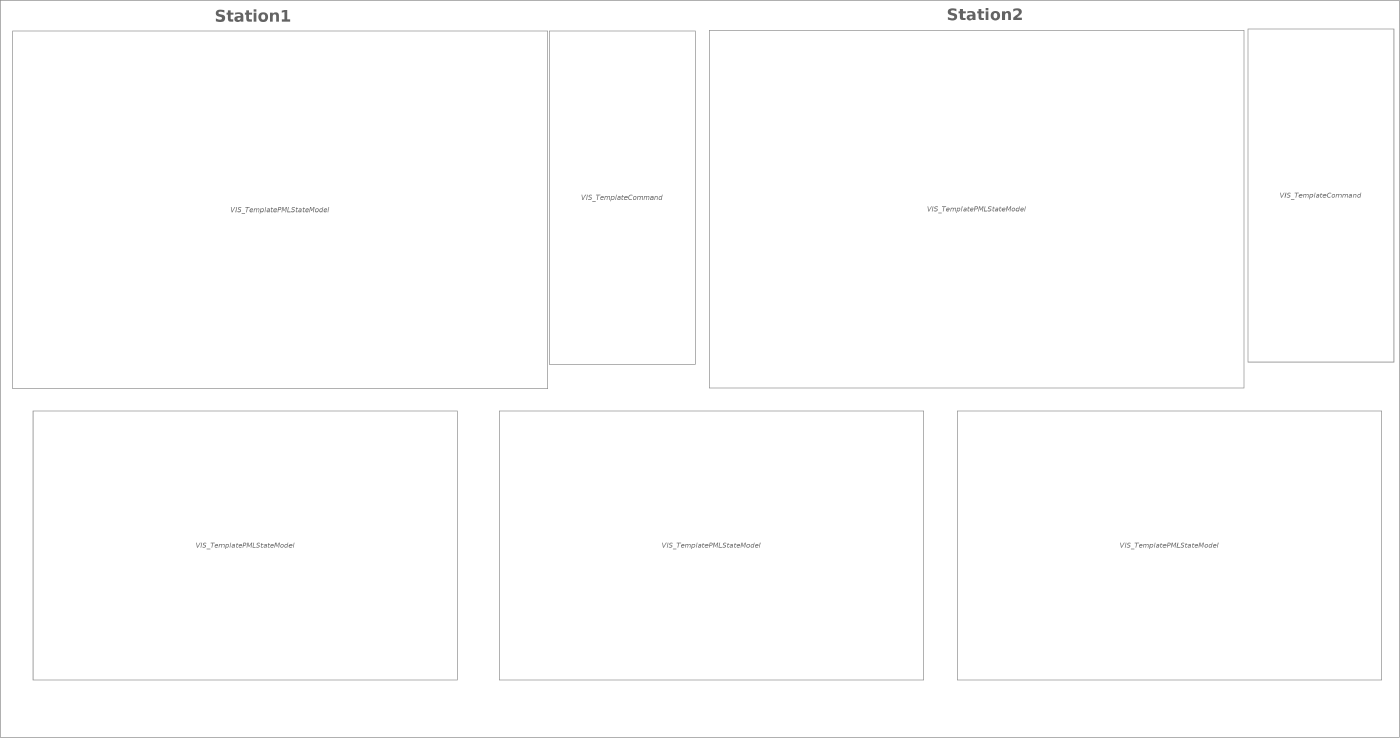
VISUALIZATION visu_2sys  // 2048x1080
    Frame (803,45 214x488)
        shows VIS_TemplateCommand(eModeCommand := GVL.PackTags.Command.UnitMode, eStateCommand := GVL.PackTags1.Command.CntrlCmd, eModeStatus := GVL.PackTags.Status.UnitModeCurrent, eStateStatus := GVL.PackTags1.Status.StateCurrent, bModeChangeReq := GVL.PackTags.Command.UnitModeChangeRequest)
    Frame (1825,42 214x488)
        shows VIS_TemplateCommand(eModeCommand := GVL.PackTags.Command.UnitMode, eStateCommand := GVL.PackTags2.Command.CntrlCmd, eModeStatus := GVL.PackTags.Status.UnitModeCurrent, eStateStatus := GVL.PackTags2.Status.StateCurrent, bModeChangeReq := GVL.PackTags.Command.UnitModeChangeRequest)
    Frame (18,45 783x524)
        shows VIS_TemplatePMLStateModel(ePMLUnitMode := MAIN.fbVisu.eModeVisu, ePMLState := MAIN.fbMachine1.eState, eStateCommand := MAIN.fbVisu.eUnitCommand)
        shows VIS_TemplatePMLStateModel()
    Frame (1037,44 783x524)
        shows VIS_TemplatePMLStateModel(ePMLUnitMode := MAIN.fbVisu.eModeVisu, ePMLState := MAIN.fbMachine2.eState, eStateCommand := MAIN.fbVisu.eUnitCommand)
        shows VIS_TemplatePMLStateModel()
    Frame (48,601 621x394)
        shows VIS_TemplatePMLStateModel(ePMLUnitMode := MAIN.fbVisu.eModeVisu, ePMLState := GVL.fb_working1.eState, eStateCommand := MAIN.fbVisu.eUnitCommand)
        shows VIS_TemplatePMLStateModel()
    Frame (730,601 621x394)
        shows VIS_TemplatePMLStateModel(ePMLUnitMode := MAIN.fbVisu.eModeVisu, ePMLState := GVL.fb_loading.eState, eStateCommand := MAIN.fbVisu.eUnitCommand)
        shows VIS_TemplatePMLStateModel()
    Frame (1400,601 621x394)
        shows VIS_TemplatePMLStateModel(ePMLUnitMode := MAIN.fbVisu.eModeVisu, ePMLState := GVL.fb_working2.eState, eStateCommand := MAIN.fbVisu.eUnitCommand)
        shows VIS_TemplatePMLStateModel()
    Label (295,1 150x45), "Station1"
    Label (1366,-1 150x45), "Station2"
END_VISUALIZATION

(* stored: Version 1.1.0.1, ProductVersion 3.1.4024.12
   Visu visu_2sys: Id {ca5e7b6f-e3a1-4c60-abe9-aa26e2843835} *)
